{attribute 'GeneratedUsingTerminal: EKM1101-0000-0016'}
{attribute addProperty BoxType "EKM1101-0000-0016"}
{attribute addProperty Id "ErrorBOOL1UnderrangeBOOL1OverrangeBOOL1DiagBOOL1Sensor_OvrBOOL1OverrunBOOL1TxPDO_StateBOOL1"}
{attribute addProperty CRC "3124567133"}
{attribute addProperty Size "7"}
TYPE Status_BA3D1C5D :
STRUCT
	{attribute addProperty Name "Error"}
	Error : BOOL;
	{attribute addProperty Name "Underrange"}
	Underrange : BOOL;
	{attribute addProperty Name "Overrange"}
	Overrange : BOOL;
	{attribute addProperty Name "Diag"}
	Diag : BOOL;
	{attribute addProperty Name "Sensor_Ovr"}
	Sensor_Ovr : BOOL;
	{attribute addProperty Name "Overrun"}
	Overrun : BOOL;
	{attribute addProperty Name "TxPDO_State"}
	TxPDO_State : BOOL;
END_STRUCT
END_TYPE

(* stored: Version 1.2.0.0, ProductVersion 3.1.4024.9
   DUT Status_BA3D1C5D: Id {7488dd97-2d97-4cc4-827c-0f1236d5d5c6} *)
